DATA_BLOCK "setpoint"
{ S7_Optimized_Access := 'FALSE' }
VERSION : 0.1
   STRUCT
      pass : DInt;
      I1_Max : DInt;
      I2_Max : DInt;
      I3_Max : DInt;
   END_STRUCT;


BEGIN

END_DATA_BLOCK

